Staubli VAL3: showPoint.pgx

program showPoint()
  local point l_pPoint[2]
  local num l_nIndexTool
  local tool l_tTool
  local point l_pHere
  local num i
  local joint l_jHere
begin
//  // check for the @ position and the ! position
//  call trajType:getPoint(l_pPoint,false,nIndex)
//  call trajType:getTool(l_nIndexTool)
//  call trajType:getFrame(fFather,false)
//  call tcp:getTool(l_tTool,l_nIndexTool)
//  l_pHere=here(l_tTool,fFather)
//  // show it
//  if isEmpty() and distance(l_pHere.trsf,l_pPoint.trsf)<0.1
//    call use:type(use:nTopX,use:nTopY+1+use:nView,"@")
//  elseIf position(l_pPoint,fFather)=={0,0,0,0,0,0}
//    call use:type(use:nTopX,use:nTopY+1+use:nView,"0")
//  elseIf distance(l_pPoint.trsf,l_pHere.trsf)<10
//    call use:type(use:nTopX,use:nTopY+1+use:nView,"~")
//  elseIf !pointToJoint(l_tTool,l_jHere,l_pPoint,l_jHere)
//    call use:type(use:nTopX,use:nTopY+1+use:nView,"!")
//  else
//    call use:type(use:nTopX,use:nTopY+1+use:nView,"│")
//  endIf
end
